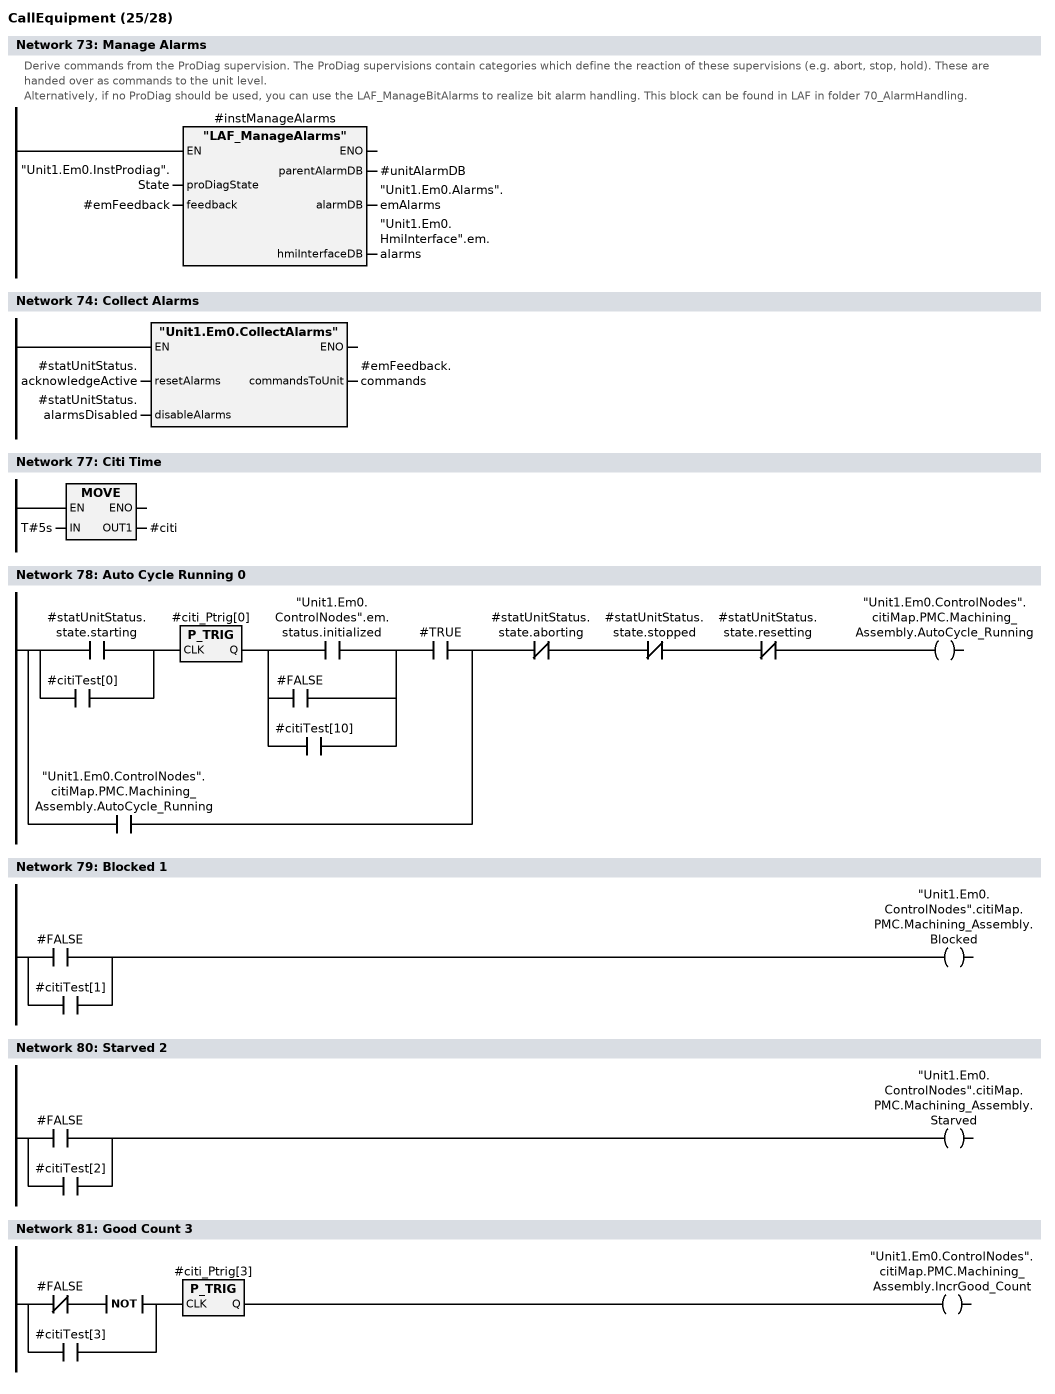
   RUNG wire#powerrail
      #instManageAlarms(proDiagState := "Unit1.Em0.InstProdiag".State, feedback := #emFeedback, parentAlarmDB => #unitAlarmDB, alarmDB => "Unit1.Em0.Alarms".emAlarms, hmiInterfaceDB => "Unit1.Em0.HmiInterface".em.alarms)
   END_RUNG
   // the same network as SCL:
   #instManageAlarms(proDiagState := "Unit1.Em0.InstProdiag".State,   // "LAF_ManageAlarms"
                     feedback := #emFeedback,
                     parentAlarmDB => #unitAlarmDB,
                     alarmDB => "Unit1.Em0.Alarms".emAlarms,
                     hmiInterfaceDB => "Unit1.Em0.HmiInterface".em.alarms);
END_REGION

REGION Network 74: Collect Alarms
   RUNG wire#powerrail
      "Unit1.Em0.CollectAlarms"(resetAlarms := #statUnitStatus.acknowledgeActive, disableAlarms := #statUnitStatus.alarmsDisabled, commandsToUnit => #emFeedback.commands)
   END_RUNG
   // the same network as SCL:
   "Unit1.Em0.CollectAlarms"(resetAlarms := #statUnitStatus.acknowledgeActive,
                           disableAlarms := #statUnitStatus.alarmsDisabled,
                           commandsToUnit => #emFeedback.commands);
END_REGION

REGION Network 76: ******************** CITI ********************
END_REGION

REGION Network 77: Citi Time
   RUNG wire#powerrail
      Move(in := T#5s, out1 => #citi)
   END_RUNG
   // the same network as SCL:
   #citi := T#5s;
END_REGION

REGION Network 78: Auto Cycle Running 0
   RUNG wire#powerrail
      Contact( #statUnitStatus.state.starting )
      wire#w1
      P_Trig( #citi_Ptrig[0] )
      wire#w2
      Contact( "Unit1.Em0.ControlNodes".em.status.initialized )
      wire#w3
      Contact( #TRUE )
      wire#w4
      I_Contact( #statUnitStatus.state.aborting )
      I_Contact( #statUnitStatus.state.stopped )
      I_Contact( #statUnitStatus.state.resetting )
      Coil( "Unit1.Em0.ControlNodes".citiMap.PMC.Machining_Assembly.AutoCycle_Running )
   END_RUNG
   RUNG wire#powerrail
      Contact( #citiTest[0] )
   END_RUNG wire#w1
   RUNG wire#w2
      Contact( #FALSE )
   END_RUNG wire#w3
   RUNG wire#w2
      Contact( #citiTest[10] )
   END_RUNG wire#w3
   RUNG wire#powerrail
      Contact( "Unit1.Em0.ControlNodes".citiMap.PMC.Machining_Assembly.AutoCycle_Running )
   END_RUNG wire#w4
   // the same network as SCL:
   #_w1 := #statUnitStatus.state.starting OR #citiTest[0];
   #_w2 := #_w1 AND NOT #citi_Ptrig[0];   // rising edge
   #citi_Ptrig[0] := #_w1;
   "Unit1.Em0.ControlNodes".citiMap.PMC.Machining_Assembly.AutoCycle_Running := ((#_w2 AND ("Unit1.Em0.ControlNodes".em.status.initialized OR #FALSE OR #citiTest[10]) AND #TRUE) OR "Unit1.Em0.ControlNodes".citiMap.PMC.Machining_Assembly.AutoCycle_Running) AND NOT #statUnitStatus.state.aborting AND NOT #statUnitStatus.state.stopped AND NOT #statUnitStatus.state.resetting;
END_REGION

REGION Network 79: Blocked 1
   RUNG wire#powerrail
      Contact( #FALSE )
      wire#w1
      Coil( "Unit1.Em0.ControlNodes".citiMap.PMC.Machining_Assembly.Blocked )
   END_RUNG
   RUNG wire#powerrail
      Contact( #citiTest[1] )
   END_RUNG wire#w1
   // the same network as SCL:
   "Unit1.Em0.ControlNodes".citiMap.PMC.Machining_Assembly.Blocked := #FALSE OR #citiTest[1];
END_REGION

REGION Network 80: Starved 2
   RUNG wire#powerrail
      Contact( #FALSE )
      wire#w1
      Coil( "Unit1.Em0.ControlNodes".citiMap.PMC.Machining_Assembly.Starved )
   END_RUNG
   RUNG wire#powerrail
      Contact( #citiTest[2] )
   END_RUNG wire#w1
   // the same network as SCL:
   "Unit1.Em0.ControlNodes".citiMap.PMC.Machining_Assembly.Starved := #FALSE OR #citiTest[2];
END_REGION

REGION Network 81: Good Count 3
   RUNG wire#powerrail
      I_Contact( #FALSE )
      Not()
      wire#w1
      P_Trig( #citi_Ptrig[3] )
      Coil( "Unit1.Em0.ControlNodes".citiMap.PMC.Machining_Assembly.IncrGood_Count )
   END_RUNG
   RUNG wire#powerrail
      Contact( #citiTest[3] )
   END_RUNG wire#w1
   // the same network as SCL:
   #_w1 := NOT (NOT #FALSE) OR #citiTest[3];
   #_w2 := #_w1 AND NOT #citi_Ptrig[3];   // rising edge
   #citi_Ptrig[3] := #_w1;
   "Unit1.Em0.ControlNodes".citiMap.PMC.Machining_Assembly.IncrGood_Count := #_w2;
END_REGION

REGION Network 82: Reject Count 4 X
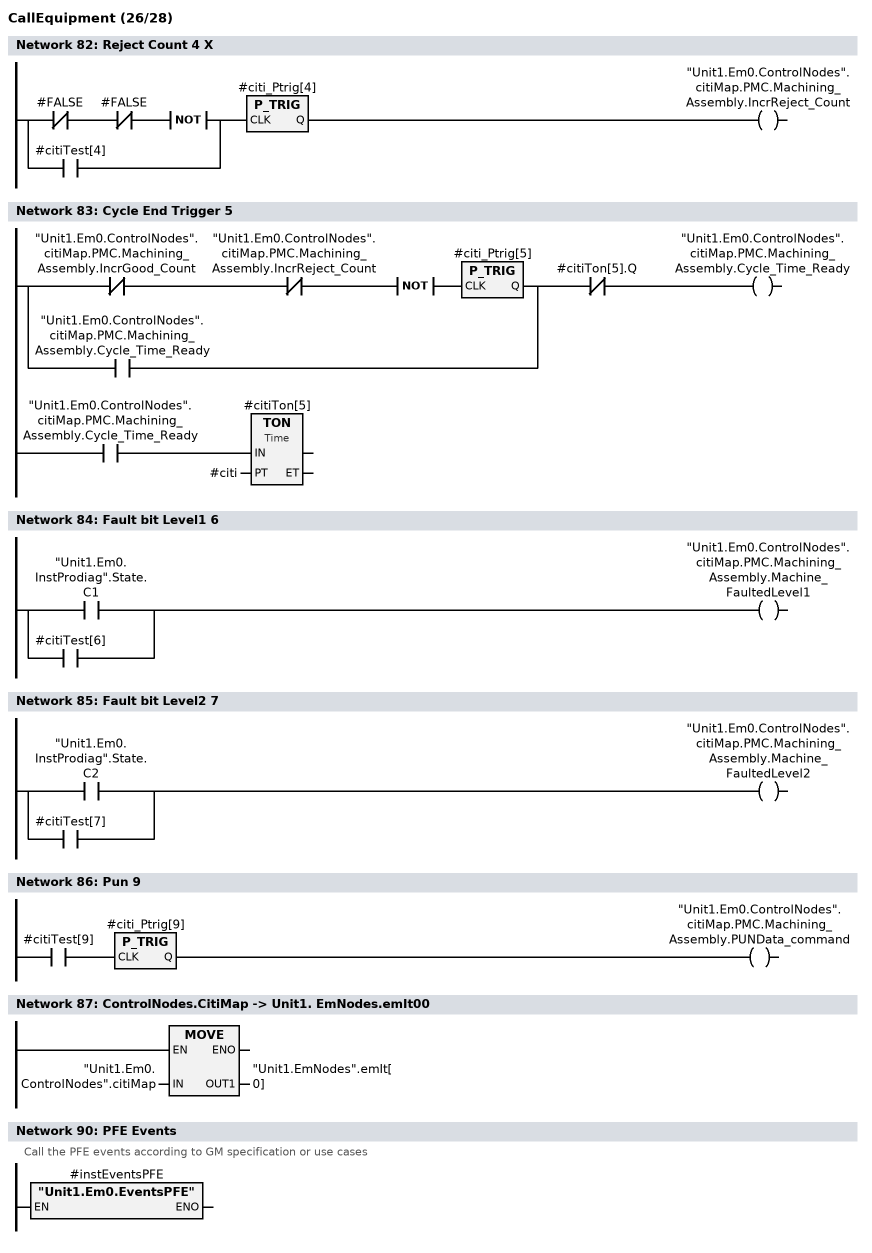
   RUNG wire#powerrail
      I_Contact( #FALSE )
      I_Contact( #FALSE )
      Not()
      wire#w1
      P_Trig( #citi_Ptrig[4] )
      Coil( "Unit1.Em0.ControlNodes".citiMap.PMC.Machining_Assembly.IncrReject_Count )
   END_RUNG
   RUNG wire#powerrail
      Contact( #citiTest[4] )
   END_RUNG wire#w1
   // the same network as SCL:
   #_w1 := NOT (NOT #FALSE AND NOT #FALSE) OR #citiTest[4];
   #_w2 := #_w1 AND NOT #citi_Ptrig[4];   // rising edge
   #citi_Ptrig[4] := #_w1;
   "Unit1.Em0.ControlNodes".citiMap.PMC.Machining_Assembly.IncrReject_Count := #_w2;
END_REGION

REGION Network 83: Cycle End Trigger 5
   RUNG wire#powerrail
      I_Contact( "Unit1.Em0.ControlNodes".citiMap.PMC.Machining_Assembly.IncrGood_Count )
      I_Contact( "Unit1.Em0.ControlNodes".citiMap.PMC.Machining_Assembly.IncrReject_Count )
      Not()
      P_Trig( #citi_Ptrig[5] )
      wire#w1
      I_Contact( #citiTon[5].Q )
      Coil( "Unit1.Em0.ControlNodes".citiMap.PMC.Machining_Assembly.Cycle_Time_Ready )
   END_RUNG
   RUNG wire#powerrail
      Contact( "Unit1.Em0.ControlNodes".citiMap.PMC.Machining_Assembly.Cycle_Time_Ready )
   END_RUNG wire#w1
   RUNG wire#powerrail
      Contact( "Unit1.Em0.ControlNodes".citiMap.PMC.Machining_Assembly.Cycle_Time_Ready )
      { S7_Templates := "time_type := Time" } #citiTon[5].TON(pt := #citi, et =>)
   END_RUNG
   // the same network as SCL:
   #_w1 := NOT (NOT "Unit1.Em0.ControlNodes".citiMap.PMC.Machining_Assembly.IncrGood_Count AND NOT "Unit1.Em0.ControlNodes".citiMap.PMC.Machining_Assembly.IncrReject_Count);
   #_w2 := #_w1 AND NOT #citi_Ptrig[5];   // rising edge
   #citi_Ptrig[5] := #_w1;
   "Unit1.Em0.ControlNodes".citiMap.PMC.Machining_Assembly.Cycle_Time_Ready := (#_w2 OR "Unit1.Em0.ControlNodes".citiMap.PMC.Machining_Assembly.Cycle_Time_Ready) AND NOT #citiTon[5].Q;
   #citiTon[5].TON(IN := "Unit1.Em0.ControlNodes".citiMap.PMC.Machining_Assembly.Cycle_Time_Ready, PT := #citi);
END_REGION

REGION Network 84: Fault bit Level1 6
   RUNG wire#powerrail
      Contact( "Unit1.Em0.InstProdiag".State.C1 )
      wire#w1
      Coil( "Unit1.Em0.ControlNodes".citiMap.PMC.Machining_Assembly.Machine_FaultedLevel1 )
   END_RUNG
   RUNG wire#powerrail
      Contact( #citiTest[6] )
   END_RUNG wire#w1
   // the same network as SCL:
   "Unit1.Em0.ControlNodes".citiMap.PMC.Machining_Assembly.Machine_FaultedLevel1 := "Unit1.Em0.InstProdiag".State.C1 OR #citiTest[6];
END_REGION

REGION Network 85: Fault bit Level2 7
   RUNG wire#powerrail
      Contact( "Unit1.Em0.InstProdiag".State.C2 )
      wire#w1
      Coil( "Unit1.Em0.ControlNodes".citiMap.PMC.Machining_Assembly.Machine_FaultedLevel2 )
   END_RUNG
   RUNG wire#powerrail
      Contact( #citiTest[7] )
   END_RUNG wire#w1
   // the same network as SCL:
   "Unit1.Em0.ControlNodes".citiMap.PMC.Machining_Assembly.Machine_FaultedLevel2 := "Unit1.Em0.InstProdiag".State.C2 OR #citiTest[7];
END_REGION

REGION Network 86: Pun 9
   RUNG wire#powerrail
      Contact( #citiTest[9] )
      P_Trig( #citi_Ptrig[9] )
      Coil( "Unit1.Em0.ControlNodes".citiMap.PMC.Machining_Assembly.PUNData_command )
   END_RUNG
   // the same network as SCL:
   #_w1 := #citiTest[9] AND NOT #citi_Ptrig[9];   // rising edge
   #citi_Ptrig[9] := #citiTest[9];
   "Unit1.Em0.ControlNodes".citiMap.PMC.Machining_Assembly.PUNData_command := #_w1;
END_REGION

REGION Network 87: ControlNodes.CitiMap -> Unit1. EmNodes.emIt00
   RUNG wire#powerrail
      Move(in := "Unit1.Em0.ControlNodes".citiMap, out1 => "Unit1.EmNodes".emIt[0])
   END_RUNG
   // the same network as SCL:
   "Unit1.EmNodes".emIt[0] := "Unit1.Em0.ControlNodes".citiMap;
END_REGION

REGION Network 89: *************** PFE Events**********************************
END_REGION

REGION Network 90: PFE Events
   // Call the PFE events according to GM specification or use cases
   RUNG wire#powerrail
      #instEventsPFE()
   END_RUNG
   // the same network as SCL:
   #instEventsPFE();   // "Unit1.Em0.EventsPFE"
END_REGION

REGION Network 91: ******************** Unit Output ********************
END_REGION

REGION Network 92: Em0 Relations SoftCam
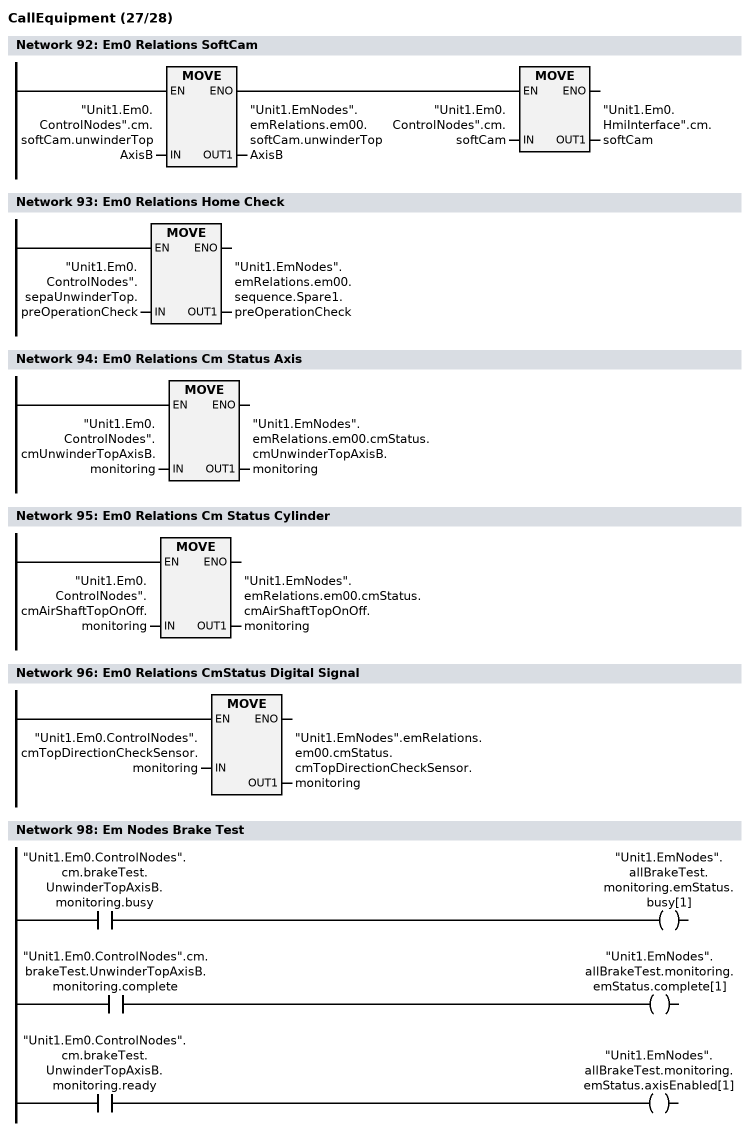
   RUNG wire#powerrail
      Move(in := "Unit1.Em0.ControlNodes".cm.softCam.unwinderTopAxisB, out1 => "Unit1.EmNodes".emRelations.em00.softCam.unwinderTopAxisB)
      Move(in := "Unit1.Em0.ControlNodes".cm.softCam, out1 => "Unit1.Em0.HmiInterface".cm.softCam)
   END_RUNG
   // the same network as SCL:
   "Unit1.EmNodes".emRelations.em00.softCam.unwinderTopAxisB := "Unit1.Em0.ControlNodes".cm.softCam.unwinderTopAxisB;
   "Unit1.Em0.HmiInterface".cm.softCam := "Unit1.Em0.ControlNodes".cm.softCam;
END_REGION

REGION Network 93: Em0 Relations Home Check
   RUNG wire#powerrail
      Move(in := "Unit1.Em0.ControlNodes".sepaUnwinderTop.preOperationCheck, out1 => "Unit1.EmNodes".emRelations.em00.sequence.Spare1.preOperationCheck)
   END_RUNG
   // the same network as SCL:
   "Unit1.EmNodes".emRelations.em00.sequence.Spare1.preOperationCheck := "Unit1.Em0.ControlNodes".sepaUnwinderTop.preOperationCheck;
END_REGION

REGION Network 94: Em0 Relations Cm Status Axis
   RUNG wire#powerrail
      Move(in := "Unit1.Em0.ControlNodes".cmUnwinderTopAxisB.monitoring, out1 => "Unit1.EmNodes".emRelations.em00.cmStatus.cmUnwinderTopAxisB.monitoring)
   END_RUNG
   // the same network as SCL:
   "Unit1.EmNodes".emRelations.em00.cmStatus.cmUnwinderTopAxisB.monitoring := "Unit1.Em0.ControlNodes".cmUnwinderTopAxisB.monitoring;
END_REGION

REGION Network 95: Em0 Relations Cm Status Cylinder
   RUNG wire#powerrail
      Move(in := "Unit1.Em0.ControlNodes".cmAirShaftTopOnOff.monitoring, out1 => "Unit1.EmNodes".emRelations.em00.cmStatus.cmAirShaftTopOnOff.monitoring)
   END_RUNG
   // the same network as SCL:
   "Unit1.EmNodes".emRelations.em00.cmStatus.cmAirShaftTopOnOff.monitoring := "Unit1.Em0.ControlNodes".cmAirShaftTopOnOff.monitoring;
END_REGION

REGION Network 96: Em0 Relations CmStatus Digital Signal
   RUNG wire#powerrail
      Move(in := "Unit1.Em0.ControlNodes".cmTopDirectionCheckSensor.monitoring, out1 => "Unit1.EmNodes".emRelations.em00.cmStatus.cmTopDirectionCheckSensor.monitoring)
   END_RUNG
   // the same network as SCL:
   "Unit1.EmNodes".emRelations.em00.cmStatus.cmTopDirectionCheckSensor.monitoring := "Unit1.Em0.ControlNodes".cmTopDirectionCheckSensor.monitoring;
END_REGION

REGION Network 97: Em0 Relations Sequence Interface
END_REGION

REGION Network 98: Em Nodes Brake Test
   RUNG wire#powerrail
      Contact( "Unit1.Em0.ControlNodes".cm.brakeTest.UnwinderTopAxisB.monitoring.busy )
      Coil( "Unit1.EmNodes".allBrakeTest.monitoring.emStatus.busy[1] )
   END_RUNG
   RUNG wire#powerrail
      Contact( "Unit1.Em0.ControlNodes".cm.brakeTest.UnwinderTopAxisB.monitoring.complete )
      Coil( "Unit1.EmNodes".allBrakeTest.monitoring.emStatus.complete[1] )
   END_RUNG
   RUNG wire#powerrail
      Contact( "Unit1.Em0.ControlNodes".cm.brakeTest.UnwinderTopAxisB.monitoring.ready )
      Coil( "Unit1.EmNodes".allBrakeTest.monitoring.emStatus.axisEnabled[1] )
   END_RUNG
   // the same network as SCL:
   "Unit1.EmNodes".allBrakeTest.monitoring.emStatus.busy[1] := "Unit1.Em0.ControlNodes".cm.brakeTest.UnwinderTopAxisB.monitoring.busy;
   "Unit1.EmNodes".allBrakeTest.monitoring.emStatus.complete[1] := "Unit1.Em0.ControlNodes".cm.brakeTest.UnwinderTopAxisB.monitoring.complete;
   "Unit1.EmNodes".allBrakeTest.monitoring.emStatus.axisEnabled[1] := "Unit1.Em0.ControlNodes".cm.brakeTest.UnwinderTopAxisB.monitoring.ready;
END_REGION

REGION Network 99 (SCL): SyncMotion Configuration
   REGION _name_
       "Unit1.MotionNodes".PLCToMotion.TechnologyObject.Axis.UnwinderTop := "Unit1.Em0.Config".axis[1];
       "Unit1.MotionNodes".PLCToMotion.Parameters.Dancer.Radius := "Unit1.Em0.ControlNodes".cmRadiusMeasure.monitoring.Radius;
       "Unit1.MotionNodes".PLCToMotion.Parameters.Dancer.UnwinderTopUse := "Unit1.EmNodes".emFeedback[0].isLinked;
   END_REGION
END_REGION

REGION Network 100: Axis
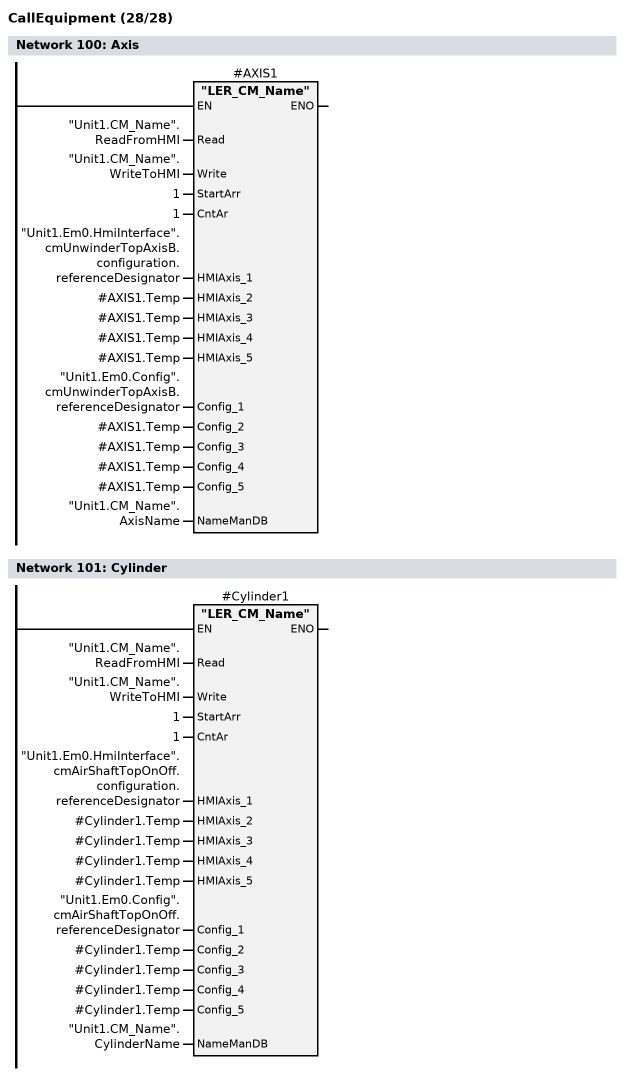
   RUNG wire#powerrail
      #AXIS1(Read := "Unit1.CM_Name".ReadFromHMI, Write := "Unit1.CM_Name".WriteToHMI, StartArr := 1, CntAr := 1, HMIAxis_1 := "Unit1.Em0.HmiInterface".cmUnwinderTopAxisB.configuration.referenceDesignator, HMIAxis_2 := #AXIS1.Temp, HMIAxis_3 := #AXIS1.Temp, HMIAxis_4 := #AXIS1.Temp, HMIAxis_5 := #AXIS1.Temp, Config_1 := "Unit1.Em0.Config".cmUnwinderTopAxisB.referenceDesignator, Config_2 := #AXIS1.Temp, Config_3 := #AXIS1.Temp, Config_4 := #AXIS1.Temp, Config_5 := #AXIS1.Temp, NameManDB := "Unit1.CM_Name".AxisName)
   END_RUNG
   // the same network as SCL:
   #AXIS1(Read := "Unit1.CM_Name".ReadFromHMI,   // "LER_CM_Name"
          Write := "Unit1.CM_Name".WriteToHMI,
          StartArr := 1,
          CntAr := 1,
          HMIAxis_1 := "Unit1.Em0.HmiInterface".cmUnwinderTopAxisB.configuration.referenceDesignator,
          HMIAxis_2 := #AXIS1.Temp,
          HMIAxis_3 := #AXIS1.Temp,
          HMIAxis_4 := #AXIS1.Temp,
          HMIAxis_5 := #AXIS1.Temp,
          Config_1 := "Unit1.Em0.Config".cmUnwinderTopAxisB.referenceDesignator,
          Config_2 := #AXIS1.Temp,
          Config_3 := #AXIS1.Temp,
          Config_4 := #AXIS1.Temp,
          Config_5 := #AXIS1.Temp,
          NameManDB := "Unit1.CM_Name".AxisName);
END_REGION

REGION Network 101: Cylinder
   RUNG wire#powerrail
      #Cylinder1(Read := "Unit1.CM_Name".ReadFromHMI, Write := "Unit1.CM_Name".WriteToHMI, StartArr := 1, CntAr := 1, HMIAxis_1 := "Unit1.Em0.HmiInterface".cmAirShaftTopOnOff.configuration.referenceDesignator, HMIAxis_2 := #Cylinder1.Temp, HMIAxis_3 := #Cylinder1.Temp, HMIAxis_4 := #Cylinder1.Temp, HMIAxis_5 := #Cylinder1.Temp, Config_1 := "Unit1.Em0.Config".cmAirShaftTopOnOff.referenceDesignator, Config_2 := #Cylinder1.Temp, Config_3 := #Cylinder1.Temp, Config_4 := #Cylinder1.Temp, Config_5 := #Cylinder1.Temp, NameManDB := "Unit1.CM_Name".CylinderName)
   END_RUNG
   // the same network as SCL:
   #Cylinder1(Read := "Unit1.CM_Name".ReadFromHMI,   // "LER_CM_Name"
              Write := "Unit1.CM_Name".WriteToHMI,
              StartArr := 1,
              CntAr := 1,
              HMIAxis_1 := "Unit1.Em0.HmiInterface".cmAirShaftTopOnOff.configuration.referenceDesignator,
              HMIAxis_2 := #Cylinder1.Temp,
              HMIAxis_3 := #Cylinder1.Temp,
              HMIAxis_4 := #Cylinder1.Temp,
              HMIAxis_5 := #Cylinder1.Temp,
              Config_1 := "Unit1.Em0.Config".cmAirShaftTopOnOff.referenceDesignator,
              Config_2 := #Cylinder1.Temp,
              Config_3 := #Cylinder1.Temp,
              Config_4 := #Cylinder1.Temp,
              Config_5 := #Cylinder1.Temp,
              NameManDB := "Unit1.CM_Name".CylinderName);
END_REGION
END_FUNCTION_BLOCK
